TYPE "Prg_GetITF"
VERSION : 0.1
// Block: Prg_GetITF
   STRUCT
      PrgNo : DInt;
      Execute : Bool;
      InProgress : Bool;
      Done : Bool;
      Error : Bool;
   END_STRUCT;

END_TYPE
